Universal Robots PolyScope program: simpleMov.urp

Program simpleMov (installation=GD directory=/home/ros/ursim-5.13.0.113898/programs createdIn=5.13.0 lastSavedIn=5.13.0 robotSerialNumber=20195299999)
Calibrated DH parameters: a=[0, -0.6127, -0.57155, 0, 0, 0]; d=[0.1807, 0, 0, 0.17415, 0.11985, 0.11655]; alpha=[1.570796, 0, 0, 1.570796, -1.570796, 0]; deltaTheta=[0, 0, 0, 0, 0, 0]
InitVariablesNode
Robot Program (runOnlyOnce=false)
  MoveJ speed 60 deg/s, acceleration 80 deg/s^2 (useActiveTCP=true) feature=Base
    Waypoint Waypoint_1: TCP in base x=541.496 y=-512.956 z=239.519 mm, rx=3.0035 ry=-0.9211 rz=0 rad; joints [-29.947, -109.118, -115.796, -45.086, 90, -85.848] deg
    Wait Sleep waitTime=1
    Waypoint Waypoint_2: TCP in base x=739.7 y=-95.839 z=591.462 mm, rx=3.1411 ry=0.0539 rz=0 rad; joints [6.12, -93.751, -94.708, -81.541, 90, -85.848] deg
    Wait Sleep waitTime=1
